{attribute addProperty BoxType "IODEVICETYPE_ETHERCATPROT"}
{attribute addProperty Id "Beckhoff_EPP1xxxBeckhoff_EPP1xxx_9DC543015440680Beckhoff_EPP2xxxBeckhoff_EPP2xxx_7FE046AD157361967Beckhoff_EPP3xxxBeckhoff_EPP3xxx_5AF4C5F17642955.25Beckhoff_EPP4xxxBeckhoff_EPP4xxx_454DDD331228153.5Beckhoff_EPP5xxxBeckhoff_EPP5xxx_36D2ADAB1442180.25Beckhoff_EPP6xxxBeckhoff_EPP6xxx_5B0359705218652.25Beckhoff_EPP7xxxBeckhoff_EPP7xxx_19C1DAAF2338292.25Beckhoff_EPP9xxxBeckhoff_EPP9xxx_B13825D253266.5SyncUnitsSyncUnits_CAB22D3B19524.375InputsInputs_C75D3FEC1280160OutputsOutputs_47D1E803848106InfoDataInfoData_E9F65A829612"}
{attribute addProperty CRC "2093016044"}
{attribute addProperty SizeInBites "41995"}
{attribute addProperty SizeInBytes "5249.375"}
TYPE EtherCAT_Master_EPPxxxx_7CC0E3EC :
STRUCT
	{attribute addProperty Name "Beckhoff_EPP1xxx"}
	Beckhoff_EPP1xxx : Beckhoff_EPP1xxx_9DC54301;
	{attribute addProperty Name "Beckhoff_EPP2xxx"}
	Beckhoff_EPP2xxx : Beckhoff_EPP2xxx_7FE046AD;
	{attribute addProperty Name "Beckhoff_EPP3xxx"}
	Beckhoff_EPP3xxx : Beckhoff_EPP3xxx_5AF4C5F1;
	{attribute addProperty Name "Beckhoff_EPP4xxx"}
	Beckhoff_EPP4xxx : Beckhoff_EPP4xxx_454DDD33;
	{attribute addProperty Name "Beckhoff_EPP5xxx"}
	Beckhoff_EPP5xxx : Beckhoff_EPP5xxx_36D2ADAB;
	{attribute addProperty Name "Beckhoff_EPP6xxx"}
	Beckhoff_EPP6xxx : Beckhoff_EPP6xxx_5B035970;
	{attribute addProperty Name "Beckhoff_EPP7xxx"}
	Beckhoff_EPP7xxx : Beckhoff_EPP7xxx_19C1DAAF;
	{attribute addProperty Name "Beckhoff_EPP9xxx"}
	Beckhoff_EPP9xxx : Beckhoff_EPP9xxx_B13825D2;
	{attribute addProperty Name "SyncUnits"}
	SyncUnits : SyncUnits_CAB22D3B;
	{attribute addProperty Name "Inputs"}
	Inputs : Inputs_C75D3FEC;
	{attribute addProperty Name "Outputs"}
	Outputs : Outputs_47D1E803;
	{attribute addProperty Name "InfoData"}
	InfoData : InfoData_E9F65A82;
END_STRUCT
END_TYPE

(* stored: Version 1.2.0.0, ProductVersion 3.1.4024.9
   DUT EtherCAT_Master_EPPxxxx_7CC0E3EC: Id {7ca02e8b-cae5-47a3-80b0-852aec650be0} *)
